FUNCTION_BLOCK "_SF_TestableSafetySensor"
{ S7_Optimized_Access := 'TRUE' }
VERSION : 0.1

BEGIN
END_FUNCTION_BLOCK

